FUNCTION_BLOCK FB_T1_DataSource IMPLEMENTS I_DataSource, I_V1_Virtual_Input_Source_1
VAR_OUTPUT
	eDataState: E_DataSourceState;
END_VAR
VAR
	_bV1_Virtual_Input: BOOL;
	_nV1_Virtual_Input_1: INT;
	_tTimestamp: ULINT;
	
	_nElements: UDINT;
	_nCurrentElement: UDINT;
	
	_nDataHandle: ULINT;
	
	fbIotSymbol_MAIN_bDinx: FB_ALY_IotSymbol_BOOL := (stConfig:= (sSymbolName:= 'MAIN.bDinx'));
	fbIotSymbol_MAIN_nAinx: FB_ALY_IotSymbol_INT := (stConfig:= (sSymbolName:= 'MAIN.nAinx'));
	
	//Target T1 = Broker:"192.168.1.10" Topic:"DefaultMainTopic/PlcStream1"
	fbStreamHelper: FB_ALY_StreamHelper;
	bConfigured: BOOL := FALSE;
	
	fbALY_GetSystemTime: FB_ALY_GetSystemTime;
END_VAR

PROPERTY bNewData : BOOL
GET
bNewData:= _nElements > 0;
END_GET
END_PROPERTY

PROPERTY bV1_Virtual_Input : BOOL
GET
bV1_Virtual_Input:= _bV1_Virtual_Input;
END_GET
END_PROPERTY

METHOD Call : BOOL
VAR
	stConfig: ST_ALY_StreamHelper_Config;
END_VAR
IF NOT fbStreamHelper.bConfigured THEN
	stConfig.nObjectID:= 16#01010010;
	stConfig.nNumInputBuffer:= 20;
	fbStreamHelper.Configure(stConfig);
END_IF

IF NOT bConfigured THEN
	//MAIN.bDinx
	fbStreamHelper.AddIotSymbol(fbIotSymbol_MAIN_bDinx);
	//MAIN.nAinx
	fbStreamHelper.AddIotSymbol(fbIotSymbol_MAIN_nAinx);

	bConfigured:= TRUE;
END_IF

fbStreamHelper.Call();
IF fbStreamHelper.bError THEN
	eDataState:= E_DataSourceState.eError;
ELSIF NOT fbStreamHelper.bConnected THEN
	eDataState:= E_DataSourceState.eNotConnected;
ELSE
	IF eDataState <> E_DataSourceState.eReceiveData_Cancel AND eDataState <> E_DataSourceState.eReceiveData_Pause THEN
		eDataState:= E_DataSourceState.eReceiveData;
		_nElements:= fbStreamHelper.nNumElements;
	ELSE
		_nElements:= 0;
	END_IF
END_IF

fbALY_GetSystemTime.Call();


IF _nElements > 0 THEN
	_nDataHandle:= _nDataHandle + 1;
END_IF

_nCurrentElement:= 0;
END_METHOD

PROPERTY dtTimestamp : DCTIMESTRUCT
GET

dtTimestamp:= F_AlyTimestampToDCTimestruct(_tTimestamp);
END_GET
END_PROPERTY

METHOD GetData : BOOL
VAR_INPUT
	nElement: UDINT;
END_VAR
VAR
END_VAR
IF nElements > 0 THEN
	IF nElement <= nElements THEN

		IF _nCurrentElement <> nElement THEN
			//Set local raw inputs
			_bV1_Virtual_Input:= fbIotSymbol_MAIN_bDinx.GetValue(nElement);
			_nV1_Virtual_Input_1:= fbIotSymbol_MAIN_nAinx.GetValue(nElement);

			//Set tTimestamp
			_tTimestamp:= fbStreamHelper.GetTimestampElement(nElement);


			_nCurrentElement:= nElement;
		END_IF
	END_IF
	GetData:= TRUE;
ELSE
	GetData:= FALSE;
END_IF
END_METHOD

METHOD HistoricalCtrl : BOOL
VAR_INPUT
	stCtrl: REFERENCE TO ST_HMI_DataSourceCtrl;
	stHistStreamInfo: REFERENCE TO ST_HMI_DataSourceHist;
	stRecordInfo: REFERENCE TO ST_HMI_DataSourceHistRecordInfo;
END_VAR
VAR
END_VAR
//Not implemented
END_METHOD

PROPERTY nDataHandle : ULINT
GET
nDataHandle:= _nDataHandle;
END_GET
END_PROPERTY

PROPERTY nElements : UDINT
GET
nElements:= _nElements;
END_GET
END_PROPERTY

METHOD NewDataAvailable : BOOL
VAR_INPUT
	nLastDataHandle: ULINT;
END_VAR
VAR
END_VAR
NewDataAvailable:= _nElements > 0 AND _nDataHandle <> nLastDataHandle;
END_METHOD

PROPERTY nV1_Virtual_Input_1 : INT
GET
nV1_Virtual_Input_1:= _nV1_Virtual_Input_1;
END_GET
END_PROPERTY

PROPERTY tTimestamp : ULINT
GET
tTimestamp:= _tTimestamp;
END_GET
END_PROPERTY

METHOD UpdateRecordList : BOOL
VAR_INPUT
	stCtrl: REFERENCE TO ST_HMI_DataSourceCtrl;
	sStreamSystemID: GUID;
	stHistStreamInfo: REFERENCE TO ST_HMI_DataSourceHist;
END_VAR
VAR
END_VAR
//Not implemented
END_METHOD

END_FUNCTION_BLOCK

(* stored: Version 1.1.0.1, ProductVersion 3.1.4024.4
   POU FB_T1_DataSource: Id {5bc0c52f-4191-4e99-a720-931412f63f26}, SpecialFunc None
   Property bNewData: Id {3fc89be7-97e2-41de-8139-98bd6fe92b28}
   Get Get: Id {5c7dd1c0-d6e1-4dec-9973-695118e14be0}
   Property bV1_Virtual_Input: Id {c17c9d2d-7d79-4b75-bd70-6ed39e0b31c8}
   Get Get: Id {ae1eaa8c-d6de-42f6-b17b-a7289613259f}
   Method Call: Id {f23b20d7-9dd6-4602-8812-48a155a318b9}
   Property dtTimestamp: Id {8719ce5e-c77c-4928-9cc6-732849c82853}
   Get Get: Id {2e6d13de-cc56-4cbe-9c0d-bd7c3554b7ec}
   Method GetData: Id {f381fa0a-f49a-4666-9869-28ccacd93091}
   Method HistoricalCtrl: Id {6166c508-6aa1-489e-a523-69b2fe447fb0}
   Property nDataHandle: Id {f97f09ad-b157-4b76-a02c-7f8c8172177f}
   Get Get: Id {d40d3f8d-b013-4ae7-bc73-f56fd026f188}
   Property nElements: Id {efbdc9e3-2881-48da-a1f5-9d0a62ac3193}
   Get Get: Id {b882c6a2-49d9-4172-9d41-e4600839da3c}
   Method NewDataAvailable: Id {11f195fa-94d4-45aa-8be9-1f0c099ab709}
   Property nV1_Virtual_Input_1: Id {a1164c13-bdf8-44d1-89b3-c161729bcb24}
   Get Get: Id {e48310d6-d488-442b-ada2-239c1420a364}
   Property tTimestamp: Id {2d75c692-cfeb-43ac-8b34-7560403e08cc}
   Get Get: Id {9596e2b4-8fa2-4fcf-bb7c-1b33603385bb}
   Method UpdateRecordList: Id {2c980400-9403-4f57-8635-a598f5a2f1d5} *)
